// Block: A02_HMI

DATA_BLOCK A02_HMI
VERSION : 0.1
   NON_RETAIN
   VAR
      Area02 : Struct
         Status : StatusArea;
         SuperUser : SuperUser;
      END_STRUCT;
      MB2 : Struct
         ManCode_REQ : Int;
         ManCode_CMD : Int;
         Button : Struct
            Area02HU : Struct
               Stop : Bool;
               Start : Bool;
            END_STRUCT;
            PitTable1 : ValveMachine_PB;
            Profilatrice_RegolazioneFormato : Struct
               Single_PB : Array[1..14] of Ax_PB;
               Passaggio02_Combo : Ax_PB;
               Passaggio14_Combo : Ax_PB;
               Passaggio17_Combo : Ax_PB;
               Passaggio18_Combo : Ax_PB;
            END_STRUCT;
            Rollformer : Struct
               Feed : Ax_PB;
               Lubr1 : Struct
                  Start : Bool;
                  Stop : Bool;
               END_STRUCT;
               Lubr2 : Struct
                  Start : Bool;
                  Stop : Bool;
               END_STRUCT;
               Lubr3 : Struct
                  Start : Bool;
                  Stop : Bool;
               END_STRUCT;
            END_STRUCT;
            MwFacCalc : Struct
               PushAx : Ax_PB;
               Gripper : ValveMachine_PB;
            END_STRUCT;
            FlyingCarriage : Struct
               Move : Ax_PB;
               Lubr : Struct
                  Start : Bool;
                  Stop : Bool;
               END_STRUCT;
               ZeroFind : Bool;
            END_STRUCT;
            FinalCut : Struct
               CutHead : ValveMachine_PB;
               DrawHead : ValveMachine_PB;
               MarkHead : ValveMachine_PB;
               Locking : ValveMachine_PB;
               Lubr : Struct
                  Start : Bool;
                  Stop : Bool;
               END_STRUCT;
            END_STRUCT;
            AccRollConveyor : Struct
               Move1 : Ax_PB;
               Move2 : Ax_PB;
               Move3 : Ax_PB;
               MoveCombo : Ax_PB;
               PusherVert_Single : Array[1..MAX_PUSHER] of ValveMachine_PB;
               PusherHoriz_Single : Array[1..MAX_PUSHER] of ValveMachine_PB;
               PusherVertCombo : ValveMachine_PB;
               PusherHorizCombo : ValveMachine_PB;
            END_STRUCT;
            PB_Empty : Struct
               Valve : ValveMachine_PB;
               Ax : Ax_PB;
            END_STRUCT;
         END_STRUCT;
      END_STRUCT;
   END_VAR

BEGIN
   // No initialization required
END_DATA_BLOCK
